FUNCTION_BLOCK Conveyor
VAR_INPUT
    // We Inject the dependency via an Interface reference
    itfMotor : GpMotor; 
END_VAR
VAR
    isStarted : BOOL;
END_VAR


IF isStarted THEN
    itfMotor.Start(); // The conveyor doesn't know IF it's a Servo or Digital!
ELSE
    itfMotor.Stop();
END_IF

END_FUNCTION_BLOCK

(* stored: Version 1.1.0.1, ProductVersion 3.1.4024.16
   POU Conveyor: Id {bd1496dd-35e8-47b4-a3a5-4c5102fbec2c}, SpecialFunc None *)
